FUNCTION_BLOCK RpcResponseManager IMPLEMENTS I_RpcResponseManager
VAR
	asyncResponses : Dictionary;
	config : I_RpcResponseManagerConfig;
END_VAR

METHOD FB_init : BOOL
VAR_INPUT
	bInitRetains : BOOL; // if TRUE, the retain variables are initialized (warm start / cold start)
	bInCopyCode : BOOL;  // if TRUE, the instance afterwards gets moved into the copy code (online change)
	Config : I_RpcResponseManagerConfig;
END_VAR
THIS^.config := Config;
END_METHOD

END_FUNCTION_BLOCK

(* stored: Version 1.1.0.1, ProductVersion 3.1.4024.12
   POU RpcResponseManager: Id {3f208033-fc55-4901-a839-41a96f923931}, SpecialFunc None
   Folder Constructor: Id {4cf791e2-033e-41c1-bd7f-0547acd5686e}
   Method FB_init: Id {53fea6ea-86b0-4213-974d-53d7704695f3} *)
